PROGRAM MAIN
VAR
END_VAR

END_PROGRAM

(* stored: Version 1.1.0.1
   POU MAIN: Id {05ca9d23-59e4-49f5-a862-51edc455695f} *)
